////////////////////////////////////////////////////////////////////////////////
      OPN   DB [#DBEventos];
      L     '[';  // Evento - Atributo Numero de Dispositivo '[LLAV]'
      T     DBB [AR2, P#0.0];
      L     'LLAV';
      T     DBD [AR2, P#1.0];
      L     ']';
      T     DBB [AR2, P#5.0];
      +AR2  P#6.0;

      L     "DB831_Mesas".Mesas[#NumMesa].StatusActual;
      L     W#16#F0;  // Solo la parte Llave
      AW;
      SRD   4;
      L     10;
      +I;
      T     #Convertir;

      T     #Convertir;
      CALL  "FC895_Obtener_EtiquetaDeValor"
      ( ValorEvento    := #Convertir,
        EtiquetaEvento := #Conversion
      );

      OPN   DB [#DBEventos];
      L     #Conversion;
      T     DBD [AR2, P#0.0];
      +AR2  P#4.0;


////////////////////////////////////////////////////////////////////////////////
      OPN   DB [#DBEventos];
      L     '[';  // Evento - Atributo Numero de Dispositivo '[HABI]'
      T     DBB [AR2, P#0.0];
      L     'HABI';
      T     DBD [AR2, P#1.0];
      L     ']';
      T     DBB [AR2, P#5.0];
      +AR2  P#6.0;

      L     2001;  // Inicializar: Decir que esta Habilitado
      T     #Convertir;

      SET;
      AN    "DB831_Mesas".Mesas[#NumMesa].Memorias.DesHabilitado;
      JC    HabilitadoDispositivo_STAT_EventosMesa;  // Esta Habilitado ??

      L     2002;
      T     #Convertir;

HabilitadoDispositivo_STAT_EventosMesa:NOP   0;
      CALL  "FC895_Obtener_EtiquetaDeValor"
      ( ValorEvento    := #Convertir,
        EtiquetaEvento := #Conversion
      );

      OPN   DB [#DBEventos];  // Se pasa al Evento
      L     #Conversion;
      T     DBW [AR2, P#0.0];
      +AR2  P#2.0;


////////////////////////////////////////////////////////////////////////////////
      OPN   DB [#DBEventos];
      L     '[';  // Evento - Atributo Numero de Dispositivo '[PRIO]'
      T     DBB [AR2, P#0.0];
      L     'PRIO';
      T     DBD [AR2, P#1.0];
      L     ']';
      T     DBB [AR2, P#5.0];
      +AR2  P#6.0;

      L     "DB831_Mesas".Mesas[#NumMesa].Prioridad;
      T     #Convertir;  // Se pasa a ASCII
      L     W#16#30;
      +I;
      T     #Convertir;

      OPN   DB [#DBEventos];  // Se pasa al Evento
      T     DBB [AR2, P#0.0];
      +AR2  P#1.0;

////////////////////////////////////////////////////////////////////////////////
// Poner Error (Si es necesario)

      L     "DB831_Mesas".Mesas[#NumMesa].ErrorActual;
      L     0;
      ==D;
      JC    SinErrorDispositivo_STAT_EventosMesa;

      L     "DB831_Mesas".Mesas[#NumMesa].ErrorActual;
      T     #Valor;

      OPN   DB [#DBEventos];
      L     '[';  // Evento - Atributo Numero de Dispositivo '[CODE]'
      T     DBB [AR2, P#0.0];
      L     'CODE';
      T     DBD [AR2, P#1.0];
      L     ']';
      T     DBB [AR2, P#5.0];
      +AR2  P#6.0;

// --- Convertir Valor a ASCII - Error
      TAR2;
      SRD   3;
      T     #NumBytes;  // Miro que offset tiene la String

      CALL  "FC893_Obtener_StringDelAtributo"
      ( DB_String := #NumDBEventos,
        OffsetIni := #NumBytes,
        Valor     := #Valor,
        OffsetFin := #Offset
      );  // Llamo a ObtenerStrinAtributo

      L     #Offset;
      SLD   3;
      LAR2;  // Recupero que offset tiene la String

// --- Ya esta convertido el Valor a ASCII

SinErrorDispositivo_STAT_EventosMesa:NOP   0;


////////////////////////////////////////////////////////////////////////////////
// Final del formaateo del Evento

      OPN   DB [#DBEventos];  // DB de Eventos Generados (A Emitir)
      L     '}';  // Fin de Evento '}'
      T     DBB [AR2, P#0.0];
      +AR2  P#1.0;


////////////////////////////////////////////////////////////////////////////////
////////////////////////////////////////////////////////////////////////////////
////////////////////////////////////////////////////////////////////////////////
// Dar por formateado el Evento

      L     0;  // Lo doy por tratado
      T     "DB831_Mesas".Mesas[#NumMesa].EstadoEmisionEvento;

      JU    FinBucle_EventosMesa;  // No existe ese tipo de Evento

// Fin del Formateo del Evento STAT
////////////////////////////////////////////////////////////////////////////////
////////////////////////////////////////////////////////////////////////////////
////////////////////////////////////////////////////////////////////////////////



NETWORK
TITLE = --- Evento de Dispositivo Mesa - Fin de Proceso - FIN!
////////////////////////////////////////////////////////////////////////////////
////////////////////////////////////////////////////////////////////////////////
////////////////////////////////////////////////////////////////////////////////
// -- Formateo del Evento FIN! (Fin del Proceso --> Reset y Paro Blando)
GenerarEvento_FIN_EventosMesa:NOP   0;

      L     #P_Eventos;
      LAR2;  // Puntero al DB de Eventos Generados

      TAR2;  // Mirar si es el primer evento de la lista
      L     0;
      ==I;
      JC    InicioBuffer_FIN_EventosMesa;  // Es el primero

      OPN   DB [#DBEventos];
      L     ',';  // Separador entre eventos ','
      T     DBB [AR2, P#0.0];
      +AR2  P#1.0;

InicioBuffer_FIN_EventosMesa:NOP   0;
      OPN   DB [#DBEventos];  // DB de Eventos Generados (A Emitir)
      L     '{';  // Inicio de Evento '{'
      T     DBB [AR2, P#0.0];
      +AR2  P#1.0;

      L     'FIN!';  // Evento 'FIN!'
      T     DBD [AR2, P#0.0];
      +AR2  P#4.0;


////////////////////////////////////////////////////////////////////////////////
      OPN   DB [#DBEventos];
      L     '[';  // Evento - Atributo Tipo '[TIPO]'
      T     DBB [AR2, P#0.0];
      L     'TIPO';
      T     DBD [AR2, P#1.0];
      L     ']';
      T     DBB [AR2, P#5.0];
      +AR2  P#6.0;

      L     60;  // Dispo Mesa
      T     #Convertir;
      CALL  "FC895_Obtener_EtiquetaDeValor"
      ( ValorEvento    := #Convertir,
        EtiquetaEvento := #Conversion
      );

      OPN   DB [#DBEventos];
      L     #Conversion;
      T     DBD [AR2, P#0.0];
      +AR2  P#4.0;


////////////////////////////////////////////////////////////////////////////////
      L     '[';  // Evento - Atributo Numero de Dispositivo '[NUME]'
      T     DBB [AR2, P#0.0];
      L     'NUME';
      T     DBD [AR2, P#1.0];
      L     ']';
      T     DBB [AR2, P#5.0];
      +AR2  P#6.0;

      L     "CTE_OffsetMesa";
      L     #NumMesa;  // Numero de Mesa
      +I;
      T     #Valor;

// --- Convertir Valor a ASCII - Numero de Maquina
      TAR2;
      SRD   3;
      T     #NumBytes;  // Miro que offset tiene la String

      CALL  "FC893_Obtener_StringDelAtributo"
      ( DB_String := #NumDBEventos,
        OffsetIni := #NumBytes,
        Valor     := #Valor,
        OffsetFin := #Offset
      );  // Llamo a ObtenerStrinAtributo

      L     #Offset;
      SLD   3;
      LAR2;  // Recupero que offset tiene la String

// --- Ya esta convertido el Valor a ASCII


////////////////////////////////////////////////////////////////////////////////
// --- Preparo para los Siguientes Atributos Proceso, Estado del Proceso

      L     22;  // Por defecto Paro Blando
      T     #Proceso;  // Que proceso es

      L     #EventoDispositivo;
      L     153;
      -I;
      T     #ResultadoProceso;  // Resultado del Proceso

      L     #EventoDispositivo;
      L     152;
      >I;
      JC    ParoBlandoProceso_EventosMesa;  // Es Proceso de Paro Balndo ?

      L     21;
      T     #Proceso;  // Que proceso es

      L     #EventoDispositivo;
      L     151;
      -I;
      T     #ResultadoProceso;  // Resultado del Proceso

// --- Continuo con el formateo del evento
ParoBlandoProceso_EventosMesa:NOP   0;


////////////////////////////////////////////////////////////////////////////////
      OPN   DB [#DBEventos];
      L     '[';  // Evento - Atributo Numero de Dispositivo '[PROC]'
      T     DBB [AR2, P#0.0];
      L     'PROC';
      T     DBD [AR2, P#1.0];
      L     ']';
      T     DBB [AR2, P#5.0];
      +AR2  P#6.0;

      L     #Proceso;
      T     #Convertir;

      CALL  "FC895_Obtener_EtiquetaDeValor"
      ( ValorEvento    := #Convertir,
        EtiquetaEvento := #Conversion
      );

      OPN   DB [#DBEventos];
      L     #Conversion;
      T     DBD [AR2, P#0.0];
      +AR2  P#4.0;


////////////////////////////////////////////////////////////////////////////////
      OPN   DB [#DBEventos];
      L     '[';  // Evento - Atributo Numero de Dispositivo '[RSLT]'
      T     DBB [AR2, P#0.0];
      L     'RSLT';
      T     DBD [AR2, P#1.0];
      L     ']';
      T     DBB [AR2, P#5.0];
      +AR2  P#6.0;

      L     #ResultadoProceso;
      L     W#16#30;  // Convertir a ASCII
      +I;

      OPN   DB [#DBEventos];
      T     DBB [AR2, P#0.0];
      +AR2  P#1.0;


////////////////////////////////////////////////////////////////////////////////
// Final del formaateo del Evento

      OPN   DB [#DBEventos];  // DB de Eventos Generados (A Emitir)
      L     '}';  // Fin de Evento '}'
      T     DBB [AR2, P#0.0];
      +AR2  P#1.0;


////////////////////////////////////////////////////////////////////////////////
////////////////////////////////////////////////////////////////////////////////
////////////////////////////////////////////////////////////////////////////////
// Dar por formateado el Evento

      L     0;  // Lo doy por tratado
      T     "DB831_Mesas".Mesas[#NumMesa].EstadoEmisionEvento;

      JU    FinBucle_EventosMesa;  // No existe ese tipo de Evento

// Fin del Formateo del Evento FIN!
////////////////////////////////////////////////////////////////////////////////
////////////////////////////////////////////////////////////////////////////////
////////////////////////////////////////////////////////////////////////////////



NETWORK
TITLE = --- Evento de Dispositivo Mesa - Peticion de Estado del Dipositivo - DIS?
////////////////////////////////////////////////////////////////////////////////
////////////////////////////////////////////////////////////////////////////////
////////////////////////////////////////////////////////////////////////////////
// -- Formateo del Evento DIS? (Peticion de Estado del Dispositivo)
GenerarEvento_DIS_EventosMesa:NOP   0;

      L     #P_Eventos;
      LAR2;  // Puntero al DB de Eventos Generados

      TAR2;  // Mirar si es el primer evento de la lista
      L     0;
      ==I;
      JC    InicioBuffer_DIS_EventosMesa;  // Es el primero

      OPN   DB [#DBEventos];
      L     ',';  // Separador entre eventos ','
      T     DBB [AR2, P#0.0];
      +AR2  P#1.0;

InicioBuffer_DIS_EventosMesa:NOP   0;
      OPN   DB [#DBEventos];  // DB de Eventos Generados (A Emitir)
      L     '{';  // Inicio de Evento '{'
      T     DBB [AR2, P#0.0];
      +AR2  P#1.0;

      L     'DIS?';  // Evento 'DIS?'
      T     DBD [AR2, P#0.0];
      +AR2  P#4.0;


////////////////////////////////////////////////////////////////////////////////
      OPN   DB [#DBEventos];
      L     '[';  // Evento - Atributo Tipo '[TIPO]'
      T     DBB [AR2, P#0.0];
      L     'TIPO';
      T     DBD [AR2, P#1.0];
      L     ']';
      T     DBB [AR2, P#5.0];
      +AR2  P#6.0;

      L     60;  // Dispo Mesa
      T     #Convertir;
      CALL  "FC895_Obtener_EtiquetaDeValor"
      ( ValorEvento    := #Convertir,
        EtiquetaEvento := #Conversion
      );

      OPN   DB [#DBEventos];
      L     #Conversion;
      T     DBD [AR2, P#0.0];
      +AR2  P#4.0;


////////////////////////////////////////////////////////////////////////////////
      L     '[';  // Evento - Atributo Numero de Dispositivo '[NUME]'
      T     DBB [AR2, P#0.0];
      L     'NUME';
      T     DBD [AR2, P#1.0];
      L     ']';
      T     DBB [AR2, P#5.0];
      +AR2  P#6.0;

      L     "CTE_OffsetMesa";
      L     #NumMesa;  // Numero de Mesa
      +I;
      T     #Valor;

// --- Convertir Valor a ASCII - Numero de Mesa
      TAR2;
      SRD   3;
      T     #NumBytes;  // Miro que offset tiene la String

      CALL  "FC893_Obtener_StringDelAtributo"
      ( DB_String := #NumDBEventos,
        OffsetIni := #NumBytes,
        Valor     := #Valor,
        OffsetFin := #Offset
      );  // Llamo a ObtenerStrinAtributo

      L     #Offset;
      SLD   3;
      LAR2;  // Recupero que offset tiene la String

// --- Ya esta convertido el Valor a ASCII


////////////////////////////////////////////////////////////////////////////////
// Final del formaateo del Evento

      OPN   DB [#DBEventos];  // DB de Eventos Generados (A Emitir)
      L     '}';  // Fin de Evento '}'
      T     DBB [AR2, P#0.0];
      +AR2  P#1.0;


////////////////////////////////////////////////////////////////////////////////
////////////////////////////////////////////////////////////////////////////////
////////////////////////////////////////////////////////////////////////////////
// Dar por formateado el Evento

      L     0;  // Lo doy por tratado
      T     "DB831_Mesas".Mesas[#NumMesa].EstadoEmisionEvento;

      JU    FinBucle_EventosMesa;  // No existe ese tipo de Evento

// Fin del Formateo del Evento DIS?
////////////////////////////////////////////////////////////////////////////////
////////////////////////////////////////////////////////////////////////////////
////////////////////////////////////////////////////////////////////////////////



NETWORK
TITLE = Fin de la función
// Se acabo
FinalFuncion:NOP   0;


END_FUNCTION
